// TwinCAT 3 PLC project Lectures
// ProgramVersion: 3.1.4024.0
// libraries:
//   Tc2_Standard, * (Beckhoff Automation GmbH)
//   Tc2_System, * (Beckhoff Automation GmbH)
//   Tc3_Module, * (Beckhoff Automation GmbH)
// project tree:
//   DUTs/ Item.TcDUT (not stored), Location.TcDUT
//   GVLs/ Automatic.TcGVL, IO.TcGVL
//   / PlcTask.TcTTO
//   POUs/ AutomaticControl.TcPOU, CountCurrentPosition.TcPOU, CountCurrentPosition1.TcPOU, Initialize.TcPOU, ManualControl.TcPOU, MAIN.TcPOU, Motor.TcPOU, MotorSelection.TcPOU, Recipe1.TcPOU, Recipe11.TcPOU, Recipe13.TcPOU, Recipe2.TcPOU, RestorePreviousAutomaticState.TcPOU, Safety1.TcPOU (not stored)
//   POUs/Lectures%27 programs/ p00_true_false.TcPOU (not stored), p01_sequential.TcPOU (not stored), p02_clock.TcPOU (not stored), p03_SR1.TcPOU (not stored), p04_latch.TcPOU (not stored), p05_posEdge.TcPOU (not stored), p06_frontDetection.TcPOU (not stored), p07_memoryCell.TcPOU (not stored), p08_counter.TcPOU (not stored), p09_timers.TcPOU (not stored), p10_directionalInterlock.TcPOU (not stored), p11_logicalFunction.TcPOU (not stored), p12_controlLight.TcPOU (not stored)
// real-time tasks:
//   TASK PlcTask1: cycle T#10ms, priority 21, ADS port 351
//   TASK PlcTask: cycle T#10ms, priority 20, ADS port 350
// I/O:
//   DEVICE Device 1 (EtherCAT), AmsNetId 172.31.192.1.2.1
//     Term 1 (EK1200) [EK1200-7000 EtherCAT Power supply (1,5A E-Bus)]
//       Term 2 (EL1859) [EL1859 8Ch. Dig. Input 24V, 3ms, 8Ch. Dig. Output 24V, 0.5A]
//       Term 3 (EL1859) [EL1859 8Ch. Dig. Input 24V, 3ms, 8Ch. Dig. Output 24V, 0.5A]
//       Term 4 (EL9011) [EL9011 End Terminal]
//   DEVICE Device 2 (NOV-DP-RAM) (disabled)
//   DEVICE Device 3 (CX7000), AmsNetId 172.31.192.1.4.1
//     Term 1 (CX7028) [CX7028-0000-0121]
//       modules: Module 1 (DIO_2x), Module 2 (Empty Module), Module 3 (DIO_2x), Module 4 (Empty Module), Module 5 (DI_2x), Module 6 (Empty Module), Module 7 (DI_2x), Module 8 (Empty Module)
// variable links:
//   Lectures/Lectures Instance <-> Device 1 (EtherCAT)/Term 1 (EK1200)/Term 2 (EL1859)
//     PlcTask Inputs/IO.EndExtensionSensor <-> Channel 3/Input
//     PlcTask Inputs/IO.EndGripSensor <-> Channel 7/Input
//     PlcTask Inputs/IO.EndLiftingSensor <-> Channel 5/Input
//     PlcTask Inputs/IO.EndRotationSensor <-> Channel 1/Input
//     PlcTask Inputs/IO.StepExtensionSwitch <-> Channel 4/Input
//     PlcTask Inputs/IO.StepGripSwitch <-> Channel 8/Input
//     PlcTask Inputs/IO.StepLiftingSwitch <-> Channel 6/Input
//     PlcTask Inputs/IO.StepRotatonSwitch <-> Channel 2/Input
//     PlcTask Outputs/IO.MotorExtension <-> Channel 12/Output
//     PlcTask Outputs/IO.MotorExtensionDirection <-> Channel 11/Output
//     PlcTask Outputs/IO.MotorGrip <-> Channel 16/Output
//     PlcTask Outputs/IO.MotorGripDirection <-> Channel 15/Output
//     PlcTask Outputs/IO.MotorLifting <-> Channel 14/Output
//     PlcTask Outputs/IO.MotorLiftingDirection <-> Channel 13/Output
//     PlcTask Outputs/IO.MotorRotation <-> Channel 10/Output
//     PlcTask Outputs/IO.MotorRotationDirection <-> Channel 9/Output
//   Lectures/Lectures Instance <-> Device 3 (CX7000)/Term 1 (CX7028)
//     PlcTask Inputs/IO.ButtonGreen <-> Module 3 (DIO_2x)/DIO_2x Input Channel 2/Input
//     PlcTask Inputs/IO.ButtonLowerLeft <-> Module 5 (DI_2x)/DI_2x Input Channel 1/Input
//     PlcTask Inputs/IO.ButtonLowerRight <-> Module 5 (DI_2x)/DI_2x Input Channel 2/Input
//     PlcTask Inputs/IO.ButtonRed <-> Module 1 (DIO_2x)/DIO_2x Input Channel 1/Input
//     PlcTask Inputs/IO.ButtonUpperLeft <-> Module 1 (DIO_2x)/DIO_2x Input Channel 2/Input
//     PlcTask Inputs/IO.ButtonUpperRight <-> Module 3 (DIO_2x)/DIO_2x Input Channel 1/Input
//     PlcTask Inputs/IO.Switch <-> Module 7 (DI_2x)/DI_2x Input Channel 1/Input
//     PlcTask Outputs/IO.LEDBlueLower <-> Module 3 (DIO_2x)/DIO_2x Output Channel 2/Output
//     PlcTask Outputs/IO.LEDBlueUpper <-> Module 1 (DIO_2x)/DIO_2x Output Channel 2/Output
//     PlcTask Outputs/IO.LEDGreen <-> Module 3 (DIO_2x)/DIO_2x Output Channel 1/Output
//     PlcTask Outputs/IO.LEDRed <-> Module 1 (DIO_2x)/DIO_2x Output Channel 1/Output

CONFIGURATION Lectures
    RESOURCE PLC ON TwinCAT3
        TASK PlcTask(INTERVAL := T#10ms, PRIORITY := 21);
        PROGRAM MAIN WITH PlcTask : MAIN;
    END_RESOURCE
END_CONFIGURATION

// ---- DUTs/Location.TcDUT
TYPE Location:
STRUCT
	rotation: REAL;	// need to get full circle number...
	lifting: REAL;	// need to get the full lift number...
	extension: REAL; // need to get the full extension number...
	grip: REAL;	// need to get the full grip number...
END_STRUCT
END_TYPE

// ---- GVLs/Automatic.TcGVL
{attribute 'qualified_only'}
VAR_GLOBAL
	MotorR: Motor;
	RCurrentlyMoving: BOOL;
	RotationPositionAuto: INT;
	RotationPositionCurrent: INT;
	SafetyRON: BOOL;
	
	MotorL: Motor;
	LCurrentlyMoving: BOOL;
	LiftingPositionAuto: INT;
	LiftingPositionCurrent: INT;
	SafetyLON: BOOL;
	
	MotorE: Motor;
	ECurrentlyMoving: BOOL;
	ExtensionPositionAuto: INT;
	ExtensionPositionCurrent: INT;
	SafetyEON: BOOL;
	
	MotorG: Motor;
	GCurrentlyMoving: BOOL;
	GripPositionAuto: INT;
	GripPositionCurrent: INT;
	SafetyGON: BOOL;
	
	AllRestored: BOOL;
END_VAR

// ---- GVLs/IO.TcGVL
{attribute 'qualified_only'}
VAR_GLOBAL
	ButtonRed AT %I*: BOOL;
	ButtonUpperRight AT %I*: BOOL;
	ButtonLowerLeft AT %I*: BOOL;
	Switch AT %I*: BOOL;
	LEDRed AT %Q*: BOOL;
	LEDGreen AT %Q*: BOOL;
	ButtonUpperLeft AT %I*: BOOL;
	ButtonGreen AT %I*: BOOL;
	ButtonLowerRight AT %I*: BOOL;
	LEDBlueUpper AT %Q*: BOOL;
	LEDBlueLower AT %Q*: BOOL;
	
	EndRotationSensor AT %I*: BOOL;
	StepRotatonSwitch AT %I*: BOOL;
	EndExtensionSensor AT %I*: BOOL;
	StepExtensionSwitch AT %I*: BOOL;
	EndLiftingSensor AT %I*: BOOL;
	StepLiftingSwitch AT %I*: BOOL;
	EndGripSensor AT %I*: BOOL;
	StepGripSwitch AT %I*: BOOL;
	MotorRotationDirection AT %Q*: BOOL;
	MotorRotation AT %Q*: BOOL;
	MotorExtensionDirection AT %Q*: BOOL;
	MotorExtension AT %Q*: BOOL;
	MotorLiftingDirection AT %Q*: BOOL;
	MotorLifting AT %Q*: BOOL;
	MotorGripDirection AT %Q*: BOOL;
	MotorGrip AT %Q*: BOOL;
	Initialized: BOOL;
	MotorDirection: INT;
	PreviousManualMode: BOOL;
END_VAR

// ---- POUs/MAIN.TcPOU
PROGRAM MAIN
VAR
	ManualControl_0: ManualControl;
	AutomaticControl_0: AutomaticControl;
END_VAR

// Initially it goes to position (0,0,0,0) and initializes motors by Initialize PRG.
// There is Safety PRG that keeps checking if motors are out of bounds.
// Motors are instantiated as global vars to retain their properties.
// CountCurrentPosition PRG is the only place where we count position using the sensors.
// RestorePreviousAutomaticState is a FB that gets execture cyclic until all the directions are set to previous positions.
// AutomaticControl FB remembers which recipe is being executed and recipe remembers its state.

// TODO:
// delay...
// ce ne dela zakomentiraj Safety
VAR // added by the converter: edge detectors and wires of the graphical bodies
    _ft1 : F_TRIG;
    _rt1 : R_TRIG;
    _w1 : BOOL;
END_VAR

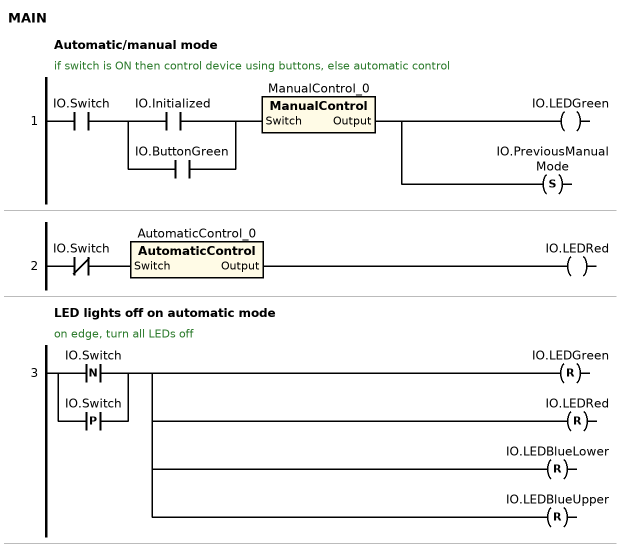
// NETWORK 1: Automatic/manual mode
// if switch is ON then control device using buttons, else automatic control
ManualControl_0(Switch := IO.Switch AND IO.Initialized OR IO.Switch AND IO.ButtonGreen); // ManualControl
IO.LEDGreen := ManualControl_0.Output;
IO.PreviousManualMode S= ManualControl_0.Output;

// NETWORK 2
AutomaticControl_0(Switch := NOT IO.Switch); // AutomaticControl
IO.LEDRed := AutomaticControl_0.Output;

// NETWORK 3: LED lights off on automatic mode
// on edge, turn all LEDs off
_ft1(CLK := IO.Switch);
_rt1(CLK := IO.Switch);
_w1 := _ft1.Q OR _rt1.Q;
IO.LEDGreen R= _w1;
IO.LEDRed R= _w1;
IO.LEDBlueLower R= _w1;
IO.LEDBlueUpper R= _w1;

END_PROGRAM

// ---- POUs/ManualControl.TcPOU
FUNCTION_BLOCK PUBLIC ManualControl
VAR_INPUT
	Switch: BOOL;
END_VAR
VAR
	ManualControl: BOOL;
	TimeForInterlockDelay: TIME := T#0.05S;
	ManualMode: BOOL;
	MotorSelection_1: MotorSelection;
	SelectedMotor: INT;
	temp: TIME;
	LowerLeftInterlock: TOF;
	LowerLeft: BOOL;
	LowerRightInterlock: TOF;
	LowerRight: BOOL;
END_VAR
VAR_OUTPUT
	Output: BOOL;
END_VAR
VAR // added by the converter: edge detectors and wires of the graphical bodies
    _w1, _w2, _w3, _w4, _w5, _w6, _w7, _w8, _w9, _w10, _w11, _w12 : BOOL;
    _rt1, _rt2, _rt3, _rt4 : R_TRIG;
    _ft1, _ft2, _ft3, _ft4 : F_TRIG;
END_VAR

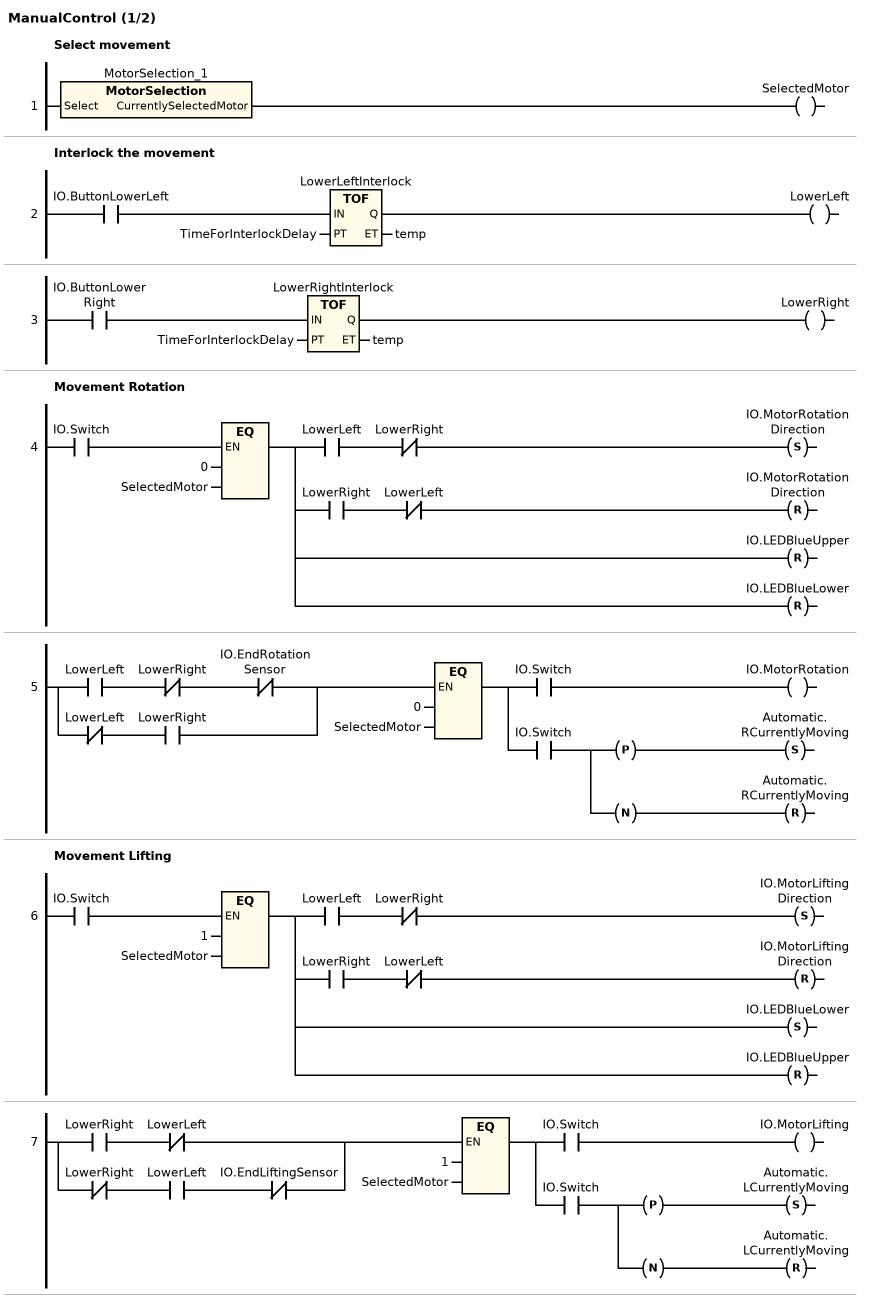
// NETWORK 1: Select movement
MotorSelection_1(Select := TRUE); // MotorSelection
SelectedMotor := MotorSelection_1.CurrentlySelectedMotor;

// NETWORK 2: Interlock the movement
LowerLeftInterlock(IN := IO.ButtonLowerLeft, PT := TimeForInterlockDelay, ET => temp); // TOF
LowerLeft := LowerLeftInterlock.Q;

// NETWORK 3
LowerRightInterlock(IN := IO.ButtonLowerRight, PT := TimeForInterlockDelay, ET => temp); // TOF
LowerRight := LowerRightInterlock.Q;

// NETWORK 4: Movement Rotation
_w1 := IO.Switch AND 0 = SelectedMotor;
IO.MotorRotationDirection S= _w1 AND LowerLeft AND NOT LowerRight;
IO.MotorRotationDirection R= _w1 AND LowerRight AND NOT LowerLeft;
IO.LEDBlueUpper R= _w1;
IO.LEDBlueLower R= _w1;

// NETWORK 5
_w2 := (LowerLeft AND NOT LowerRight AND NOT IO.EndRotationSensor OR NOT LowerLeft AND LowerRight) AND 0 = SelectedMotor;
IO.MotorRotation := _w2 AND IO.Switch;
_w3 := _w2 AND IO.Switch;
_rt1(CLK := _w3);
Automatic.RCurrentlyMoving S= _rt1.Q;
_ft1(CLK := _w3);
Automatic.RCurrentlyMoving R= _ft1.Q;

// NETWORK 6: Movement Lifting
_w4 := IO.Switch AND 1 = SelectedMotor;
IO.MotorLiftingDirection S= _w4 AND LowerLeft AND NOT LowerRight;
IO.MotorLiftingDirection R= _w4 AND LowerRight AND NOT LowerLeft;
IO.LEDBlueLower S= _w4;
IO.LEDBlueUpper R= _w4;

// NETWORK 7
_w5 := (LowerRight AND NOT LowerLeft OR NOT LowerRight AND LowerLeft AND NOT IO.EndLiftingSensor) AND 1 = SelectedMotor;
IO.MotorLifting := _w5 AND IO.Switch;
_w6 := _w5 AND IO.Switch;
_rt2(CLK := _w6);
Automatic.LCurrentlyMoving S= _rt2.Q;
_ft2(CLK := _w6);
Automatic.LCurrentlyMoving R= _ft2.Q;

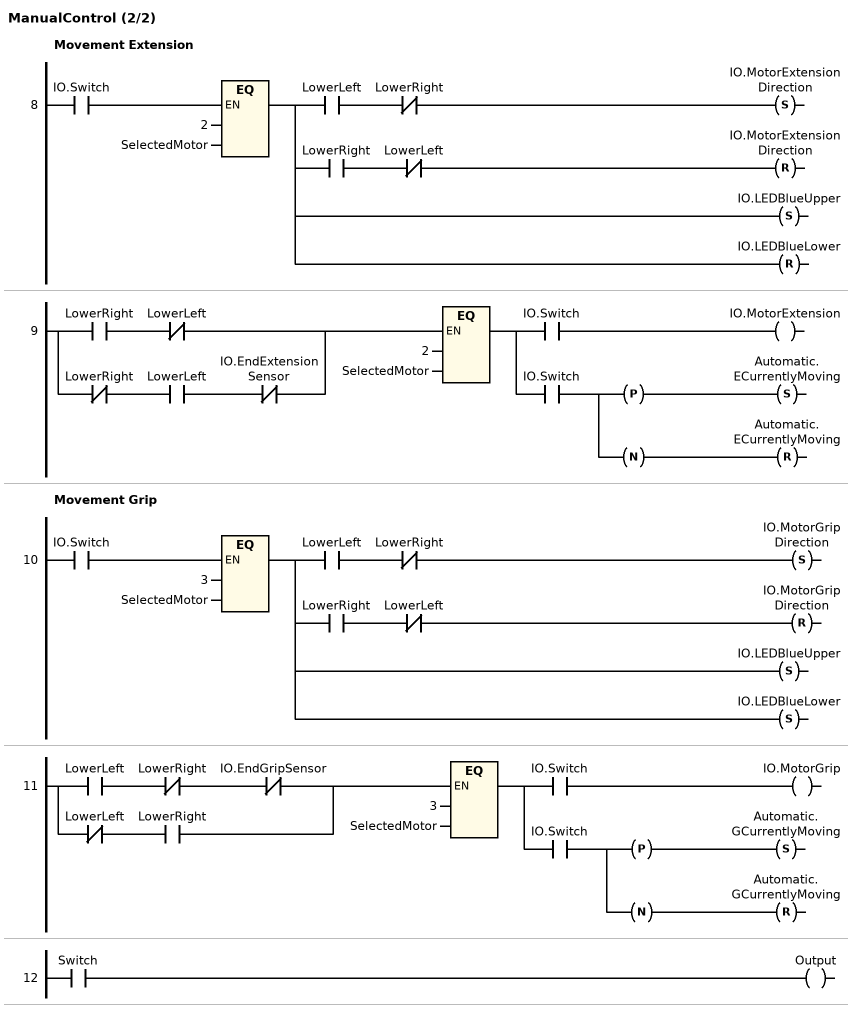
// NETWORK 8: Movement Extension
_w7 := IO.Switch AND 2 = SelectedMotor;
IO.MotorExtensionDirection S= _w7 AND LowerLeft AND NOT LowerRight;
IO.MotorExtensionDirection R= _w7 AND LowerRight AND NOT LowerLeft;
IO.LEDBlueUpper S= _w7;
IO.LEDBlueLower R= _w7;

// NETWORK 9
_w8 := (LowerRight AND NOT LowerLeft OR NOT LowerRight AND LowerLeft AND NOT IO.EndExtensionSensor) AND 2 = SelectedMotor;
IO.MotorExtension := _w8 AND IO.Switch;
_w9 := _w8 AND IO.Switch;
_rt3(CLK := _w9);
Automatic.ECurrentlyMoving S= _rt3.Q;
_ft3(CLK := _w9);
Automatic.ECurrentlyMoving R= _ft3.Q;

// NETWORK 10: Movement Grip
_w10 := IO.Switch AND 3 = SelectedMotor;
IO.MotorGripDirection S= _w10 AND LowerLeft AND NOT LowerRight;
IO.MotorGripDirection R= _w10 AND LowerRight AND NOT LowerLeft;
IO.LEDBlueUpper S= _w10;
IO.LEDBlueLower S= _w10;

// NETWORK 11
_w11 := (LowerLeft AND NOT LowerRight AND NOT IO.EndGripSensor OR NOT LowerLeft AND LowerRight) AND 3 = SelectedMotor;
IO.MotorGrip := _w11 AND IO.Switch;
_w12 := _w11 AND IO.Switch;
_rt4(CLK := _w12);
Automatic.GCurrentlyMoving S= _rt4.Q;
_ft4(CLK := _w12);
Automatic.GCurrentlyMoving R= _ft4.Q;

// NETWORK 12
Output := Switch;

END_FUNCTION_BLOCK

// ---- POUs/MotorSelection.TcPOU
FUNCTION_BLOCK PUBLIC MotorSelection
VAR_INPUT
	Select: BOOL;
END_VAR
VAR
	TimeForDelay: TIME := T#0.15S;
	MovementSelection: CTUD;
	SelectionCounter: CTUD := (LOAD := TRUE, PV := 3);
	ReachedMaxSelection: BOOL;
	ReachedMinSelection: BOOL;
	UpperLeftDelay: TOF;
	UpperRightDelay: TOF;
	tmnp: TIME;
	CU: BOOL;
	CD: BOOL;
	CUU: BOOL;
	CDD: BOOL;
	PositiveEdge1: R_TRIG;
	PositiveEdge2: R_TRIG;
	temporary: BOOL;
	CUU0: BOOL;
	CDD0: BOOL;
	temporary1: BOOL;
	BURpositiveEdge: BOOL;
	BULpositiveEdge: BOOL;
	temp2: BOOL;
	temp3: BOOL;
END_VAR
VAR_OUTPUT
	CurrentlySelectedMotor: INT;
END_VAR
VAR // added by the converter: edge detectors and wires of the graphical bodies
    _rt1, _rt2, _rt3, _rt4 : R_TRIG;
END_VAR

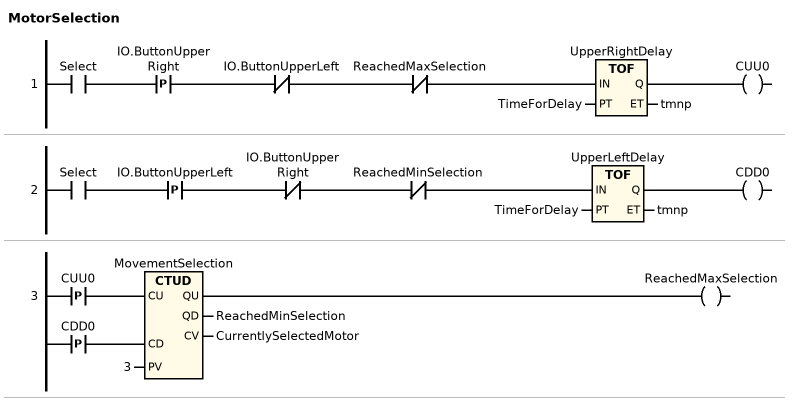
// NETWORK 1
_rt1(CLK := IO.ButtonUpperRight);
UpperRightDelay(
    IN := Select AND _rt1.Q AND NOT IO.ButtonUpperLeft AND NOT ReachedMaxSelection,
    PT := TimeForDelay,
    ET => tmnp); // TOF
CUU0 := UpperRightDelay.Q;

// NETWORK 2
_rt2(CLK := IO.ButtonUpperLeft);
UpperLeftDelay(
    IN := Select AND _rt2.Q AND NOT IO.ButtonUpperRight AND NOT ReachedMinSelection,
    PT := TimeForDelay,
    ET => tmnp); // TOF
CDD0 := UpperLeftDelay.Q;

// NETWORK 3
_rt3(CLK := CUU0);
_rt4(CLK := CDD0);
MovementSelection(
    CU := _rt3.Q,
    CD := _rt4.Q,
    PV := 3,
    QD => ReachedMinSelection,
    CV => CurrentlySelectedMotor); // CTUD
ReachedMaxSelection := MovementSelection.QU;

END_FUNCTION_BLOCK

// ---- POUs/AutomaticControl.TcPOU
FUNCTION_BLOCK PUBLIC AutomaticControl
VAR_INPUT
    Switch: BOOL;
END_VAR
VAR
    State: INT := 0;
    ExecutingRecipe1: BOOL := FALSE;
    ExecutingRecipe2: BOOL := FALSE;
    myRecipe2: Recipe2;
    Tmp: BOOL;
    RestorePreviousAutomaticState: RestorePreviousAutomaticState;
	CountCurrentPosition1: CountCurrentPosition1;
	Safety: Safety1;
END_VAR
VAR_OUTPUT
    Output: BOOL := TRUE;
END_VAR

// TwinCAT ensures that all POUs, including your AutomaticControl program 
// and Recipe1() Function Block, are executed once per cycle.

IF NOT IO.Initialized THEN
	Initialize();
ELSIF NOT IO.Switch AND IO.PreviousManualMode THEN
	Automatic.AllRestored := FALSE;
	CountCurrentPosition1();
    RestorePreviousAutomaticState();
	Safety();
ELSE
	CountCurrentPosition1();
	Safety();
	
    IF (IO.ButtonUpperLeft OR ExecutingRecipe1) AND Automatic.AllRestored THEN
		//Automatic.AllRestored := FALSE;
        ExecutingRecipe1 := TRUE;
		Recipe1();
        ExecutingRecipe1 := NOT Recipe1.SuccesfullyEnded; // Update ExecutingRecipe1 based on output
    ELSIF NOT ExecutingRecipe1 AND (IO.ButtonUpperRight OR ExecutingRecipe2) THEN
        ExecutingRecipe2 := TRUE;
        myRecipe2.ExecutingRecipe2 := ExecutingRecipe2; // Pass input to the function block
        //myRecipe2(); // Call the function block
        ExecutingRecipe2 := NOT myRecipe2.SuccesfullyEnded; // Update ExecutingRecipe2 based on output
    END_IF
END_IF


// for debugging purposes:
IF IO.ButtonRed THEN
	IO.Initialized := FALSE;
END_IF

RETURN;

END_FUNCTION_BLOCK

// ---- POUs/Recipe2.TcPOU
FUNCTION_BLOCK PUBLIC Recipe2
VAR_INPUT
	ExecutingRecipe2: BOOL;
END_VAR
VAR_OUTPUT
	SuccesfullyEnded: BOOL := FALSE;
END_VAR
VAR
	State: INT := 0;
	InitialRotationPosition: INT := 140;
	InitialLiftingPosition: INT := 200;
	MaxGripPosition: INT := 160;
END_VAR

// Recipe is sequence of moves to execute the task.

IF ExecutingRecipe2 THEN	// we start executing recipe2 (again)
	SuccesfullyEnded := FALSE;
END_IF

IF NOT IO.Switch AND NOT SuccesfullyEnded THEN
	// WOOD:
	IF State = 0 THEN
		IF Automatic.RotationPositionAuto < InitialRotationPosition THEN
			IO.MotorRotationDirection := 0;
			IF NOT Automatic.SafetyRON THEN
				Automatic.MotorR.CurrentlyMoving := TRUE;
				IO.MotorRotation := 1;
			END_IF
		ELSE
			State := 1;
			IO.MotorRotation := 0;
			Automatic.MotorR.CurrentlyMoving := FALSE;
		END_IF
	ELSIF State = 1 THEN
		IF Automatic.LiftingPositionAuto < InitialLiftingPosition THEN
			IO.MotorLiftingDirection := 1;
			IF NOT Automatic.SafetyLON THEN
				Automatic.MotorL.CurrentlyMoving := TRUE;
				IO.MotorLifting := 1;
			END_IF
		ELSE
			State := 2;
			IO.MotorLifting := 0;
			Automatic.MotorL.CurrentlyMoving := FALSE;
		END_IF
	ELSIF State = 2 THEN
		IF Automatic.GripPositionAuto < MaxGripPosition THEN
			IO.MotorGripDirection := 0;
			IF NOT Automatic.SafetyGON THEN
				Automatic.MotorG.CurrentlyMoving := TRUE;
				IO.MotorGrip := 1;
			END_IF
		ELSE
			State := 3;
			IO.MotorGrip := 0;
			Automatic.MotorG.CurrentlyMoving := FALSE;
		END_IF
	ELSIF State = 3 THEN
		IF NOT IO.EndLiftingSensor THEN
			IO.MotorLiftingDirection := 0;
			IF NOT Automatic.SafetyLON THEN
				Automatic.MotorG.CurrentlyMoving := TRUE;
				IO.MotorLifting := 1;
			END_IF
		ELSE
			State := 4;
			IO.MotorLifting := 0;
			Automatic.MotorG.CurrentlyMoving := FALSE;
		END_IF
	ELSIF State = 4 THEN
		IF NOT IO.EndRotationSensor THEN
			IO.MotorRotationDirection := 1;
			IF NOT Automatic.SafetyRON THEN
				Automatic.MotorR.CurrentlyMoving := TRUE;
				IO.MotorRotation := 1;
			END_IF
		ELSE
			State := 5;
			IO.MotorRotation := 0;
			Automatic.MotorR.CurrentlyMoving := FALSE;
		END_IF
	ELSIF State = 5 THEN
		IF NOT IO.EndGripSensor THEN		// it places the cylinder onto the platform
			IO.MotorGripDirection := 1;
			IF NOT Automatic.SafetyGON THEN
				Automatic.MotorG.CurrentlyMoving := TRUE;
				IO.MotorGrip := 1;
			END_IF
		ELSE
			State := 6;
			IO.MotorGrip := 0;
			Automatic.MotorG.CurrentlyMoving := FALSE;
		END_IF
	ELSIF State = 6 THEN
		SuccesfullyEnded := TRUE;
		State := 0;
		RETURN;
	END_IF
END_IF

END_FUNCTION_BLOCK

// ---- POUs/RestorePreviousAutomaticState.TcPOU
FUNCTION_BLOCK PUBLIC RestorePreviousAutomaticState
VAR_INPUT
END_VAR
VAR_OUTPUT
END_VAR
VAR
	RotationRestored: BOOL := FALSE;
	LiftingRestored: BOOL := FALSE;
	ExtensionRestored: BOOL := FALSE;
	GripRestored: BOOL := FALSE;
END_VAR

// reset rotation:
IO.LEDRed := 1;
IF Automatic.RotationPositionAuto - Automatic.RotationPositionCurrent > 5 AND NOT RotationRestored AND NOT Automatic.SafetyRON THEN
	IO.MotorRotationDirection := 0;
	Automatic.RCurrentlyMoving := TRUE;
	IO.MotorRotation := 1;
ELSIF Automatic.RotationPositionCurrent - Automatic.RotationPositionAuto > 5 AND NOT RotationRestored AND NOT Automatic.SafetyRON THEN
	IO.MotorRotationDirection := 1;
	Automatic.RCurrentlyMoving := TRUE;
	IO.MotorRotation := 1;
ELSE
	Automatic.RCurrentlyMoving := FALSE;
	IO.MotorRotation := 0;
	RotationRestored := TRUE;
END_IF

// reset lifting:
IF Automatic.LiftingPositionAuto - Automatic.LiftingPositionCurrent > 5 AND NOT LiftingRestored AND NOT Automatic.SafetyLON THEN
	IO.MotorLiftingDirection := 0;
	Automatic.LCurrentlyMoving := TRUE;
	IO.MotorLifting := 1;
ELSIF Automatic.LiftingPositionCurrent - Automatic.LiftingPositionAuto > 5 AND NOT LiftingRestored AND NOT Automatic.SafetyLON THEN
	IO.MotorLiftingDirection := 0;
	Automatic.LCurrentlyMoving := TRUE;
	IO.MotorLifting := 1;
ELSE
	Automatic.LCurrentlyMoving := FALSE;
	IO.MotorLifting := 0;
	LiftingRestored := TRUE;
END_IF

// reset extension:
IF Automatic.ExtensionPositionAuto - Automatic.ExtensionPositionCurrent > 5 AND NOT ExtensionRestored AND NOT Automatic.SafetyEON THEN
	IO.MotorExtensionDirection := 0;
	Automatic.ECurrentlyMoving := TRUE;
	IO.MotorExtension := 1;
ELSIF Automatic.ExtensionPositionCurrent - Automatic.ExtensionPositionAuto > 5 AND NOT ExtensionRestored AND NOT Automatic.SafetyEON THEN
	IO.MotorExtensionDirection := 0;
	Automatic.ECurrentlyMoving := TRUE;
	IO.MotorExtension := 1;
ELSE
	Automatic.ECurrentlyMoving := FALSE;
	IO.MotorExtension := 0;
	ExtensionRestored := TRUE;
END_IF

// reset grip:
IF Automatic.GripPositionAuto - Automatic.GripPositionCurrent > 5 AND NOT GripRestored AND NOT Automatic.SafetyGON THEN
	IO.MotorGripDirection := 0;
	Automatic.GCurrentlyMoving := TRUE;
	IO.MotorGrip := 1;
ELSIF Automatic.GripPositionCurrent - Automatic.GripPositionAuto > 5 AND NOT GripRestored AND NOT Automatic.SafetyGON THEN
	IO.MotorGripDirection := 0;
	Automatic.GCurrentlyMoving := TRUE;
	IO.MotorGrip := 1;
ELSE
	Automatic.GCurrentlyMoving := FALSE;
	IO.MotorGrip := 0;
	GripRestored := TRUE;
END_IF

// if all restored then go on to exeecute recipes in AutomaticControl:
IF RotationRestored AND LiftingRestored AND ExtensionRestored AND GripRestored THEN
	IO.LEDRed := 0;
	IO.PreviousManualMode := FALSE;
	Automatic.AllRestored := TRUE;
	RotationRestored := FALSE;
	ExtensionRestored := FALSE;
	LiftingRestored := FALSE;
	GripRestored := FALSE;
	Automatic.RCurrentlyMoving := FALSE;
	Automatic.ECurrentlyMoving := FALSE;
	Automatic.LCurrentlyMoving := FALSE;
	Automatic.GCurrentlyMoving := FALSE;
END_IF

END_FUNCTION_BLOCK

// ---- POUs/CountCurrentPosition1.TcPOU
FUNCTION_BLOCK CountCurrentPosition1
VAR_INPUT
END_VAR
VAR_OUTPUT
END_VAR
VAR
END_VAR

// COUNT ROTATION:
IF IO.Initialized AND IO.StepRotatonSwitch = 1 THEN
	IF IO.MotorRotationDirection = 0 THEN
		IF (NOT IO.Switch) AND Automatic.RCurrentlyMoving THEN
			IF IO.PreviousManualMode THEN
				Automatic.RotationPositionCurrent := Automatic.RotationPositionCurrent + 1;
			ELSE
				Automatic.RotationPositionCurrent := Automatic.RotationPositionCurrent + 1;
				Automatic.RotationPositionAuto := Automatic.RotationPositionAuto + 1;
			END_IF
		ELSIF Automatic.RCurrentlyMoving THEN
			Automatic.RotationPositionCurrent := Automatic.RotationPositionCurrent + 1;
		END_IF
	ELSE
		IF (NOT IO.Switch) AND Automatic.RCurrentlyMoving THEN
			IF IO.PreviousManualMode THEN
				Automatic.RotationPositionCurrent := Automatic.RotationPositionCurrent - 1;
			ELSE
				Automatic.RotationPositionCurrent := Automatic.RotationPositionCurrent - 1;
				Automatic.RotationPositionAuto := Automatic.RotationPositionAuto - 1;
			END_IF
		ELSIF Automatic.RCurrentlyMoving THEN
			Automatic.RotationPositionCurrent := Automatic.RotationPositionCurrent - 1;
		END_IF
	END_IF
END_IF

// COUNT Extension:
IF IO.Initialized AND IO.StepExtensionSwitch = 1 THEN
	IO.LEDGreen := 0;
	IF IO.MotorExtensionDirection = 0 THEN
		IF (NOT IO.Switch) AND Automatic.ECurrentlyMoving THEN
			IF IO.PreviousManualMode THEN
				Automatic.ExtensionPositionCurrent := Automatic.ExtensionPositionCurrent + 1;
			ELSE
				Automatic.ExtensionPositionAuto := Automatic.ExtensionPositionAuto + 1;
				Automatic.ExtensionPositionCurrent := Automatic.ExtensionPositionCurrent + 1;
			END_IF
		ELSIF Automatic.ECurrentlyMoving THEN
			Automatic.ExtensionPositionCurrent := Automatic.ExtensionPositionCurrent + 1;
		END_IF
	ELSE
		IF (NOT IO.Switch) AND Automatic.ECurrentlyMoving THEN
			IF IO.PreviousManualMode THEN
				Automatic.ExtensionPositionCurrent := Automatic.ExtensionPositionCurrent - 1;
			ELSE
				Automatic.ExtensionPositionAuto := Automatic.ExtensionPositionAuto - 1;
				Automatic.ExtensionPositionCurrent := Automatic.ExtensionPositionCurrent - 1;
			END_IF
		ELSIF Automatic.ECurrentlyMoving THEN
			Automatic.ExtensionPositionCurrent := Automatic.ExtensionPositionCurrent - 1;
		END_IF
	END_IF
END_IF

// COUNT Lifting:
IF IO.Initialized AND IO.StepLiftingSwitch = 1 THEN
	IF IO.MotorLiftingDirection = 0 THEN
		IF (NOT IO.Switch) AND Automatic.LCurrentlyMoving THEN
			IF IO.PreviousManualMode THEN
				Automatic.LiftingPositionCurrent := Automatic.LiftingPositionCurrent + 1;
			ELSE
				Automatic.LiftingPositionCurrent := Automatic.LiftingPositionCurrent + 1;
				Automatic.LiftingPositionAuto := Automatic.LiftingPositionAuto + 1;
			END_IF
		ELSIF Automatic.LCurrentlyMoving THEN
			Automatic.LiftingPositionCurrent := Automatic.LiftingPositionCurrent + 1;
		END_IF
	ELSE
		IF (NOT IO.Switch) AND Automatic.LCurrentlyMoving THEN
			IF IO.PreviousManualMode THEN
				Automatic.LiftingPositionCurrent := Automatic.LiftingPositionCurrent - 1;
			ELSE
				Automatic.LiftingPositionAuto := Automatic.LiftingPositionAuto - 1;
				Automatic.LiftingPositionCurrent := Automatic.LiftingPositionCurrent - 1;
			END_IF
		ELSIF Automatic.LCurrentlyMoving THEN
			Automatic.LiftingPositionCurrent := Automatic.LiftingPositionCurrent - 1;
		END_IF
	END_IF
END_IF

// COUNT Grip:
IF IO.Initialized AND IO.StepGripSwitch = 1 THEN
	IF IO.MotorGripDirection = 0 THEN
		IF (NOT IO.Switch) AND Automatic.GCurrentlyMoving THEN	// automatic mode
			IO.LEDGreen := 0;
			
			IF IO.PreviousManualMode THEN
				Automatic.GripPositionCurrent := Automatic.GripPositionCurrent + 1;
			ELSE
				Automatic.GripPositionAuto := Automatic.GripPositionAuto + 1;
				Automatic.GripPositionCurrent := Automatic.GripPositionCurrent + 1;
			END_IF
		ELSIF Automatic.GCurrentlyMoving THEN		// manual mode
			Automatic.GripPositionCurrent := Automatic.GripPositionCurrent + 1;
		END_IF
	ELSE
		IF (NOT IO.Switch) AND Automatic.GCurrentlyMoving THEN
			IO.LEDGreen := 1;
			IF IO.PreviousManualMode THEN
				Automatic.GripPositionCurrent := Automatic.GripPositionCurrent - 1;
			ELSE
				Automatic.GripPositionAuto := Automatic.GripPositionAuto - 1;
				Automatic.GripPositionCurrent := Automatic.GripPositionCurrent - 1;
			END_IF
		ELSIF Automatic.GCurrentlyMoving THEN
			Automatic.GripPositionCurrent := Automatic.GripPositionCurrent - 1;
		END_IF
	END_IF
END_IF

END_FUNCTION_BLOCK

// ---- POUs/Initialize.TcPOU
PROGRAM Initialize
VAR
END_VAR

// go to the initial position (0,0,0,0)
IF NOT IO.Initialized THEN
	IF IO.EndRotationSensor THEN
		IO.MotorRotation := 0;
		IO.MotorRotationDirection := 0;
		Automatic.MotorR.CurrentlyMoving := FALSE;
	ELSE 
		IO.MotorRotationDirection := 1;
		Automatic.MotorR.CurrentlyMoving := TRUE;
		IO.MotorRotation := 1;
	END_IF
	
	IF IO.EndLiftingSensor THEN
		IO.MotorLifting := 0;
		IO.MotorLiftingDirection := 0;
		Automatic.MotorL.CurrentlyMoving := FALSE;
	ELSE 
		IO.MotorLiftingDirection := 1;
		Automatic.MotorL.CurrentlyMoving := TRUE;
		IO.MotorLifting := 1;
	END_IF
	
	IF IO.EndExtensionSensor THEN
		IO.MotorExtension := 0;
		IO.MotorExtensionDirection := 0;
		Automatic.MotorE.CurrentlyMoving := FALSE;
	ELSE 
		IO.MotorExtensionDirection := 1;
		Automatic.MotorE.CurrentlyMoving := TRUE;
		IO.MotorExtension := 1;
	END_IF
	
	IF IO.EndGripSensor THEN
		IO.MotorGrip := 0;
		IO.MotorGripDirection := 0;
		Automatic.MotorG.CurrentlyMoving := FALSE;
	ELSE 
		IO.MotorGripDirection := 1;
		Automatic.MotorG.CurrentlyMoving := TRUE;
		IO.MotorGrip := 1;
	END_IF
		
	IF IO.EndRotationSensor AND IO.EndLiftingSensor AND IO.EndExtensionSensor AND IO.EndGripSensor THEN
		Automatic.MotorR.CurrentlyMoving := FALSE;
		Automatic.MotorE.CurrentlyMoving := FALSE;
		Automatic.MotorL.CurrentlyMoving := FALSE;
		Automatic.MotorG.CurrentlyMoving := FALSE;
		IO.Initialized := TRUE;
	END_IF
END_IF

END_PROGRAM

// ---- POUs/Recipe1.TcPOU
FUNCTION_BLOCK PUBLIC Recipe1
VAR_INPUT
	ExecutingRecipe1: BOOL;
END_VAR
VAR_OUTPUT
	SuccesfullyEnded: BOOL := FALSE;
END_VAR
VAR
	State: INT := 0;
	WoodInitialLiftingPosition: INT := 50;
	InitialExtensionPosition: INT := 388;
	MaxGripPosition: INT := 160;
	RotationDropOffPosition: INT := 300;
	PlasticsInitialLiftingPosition: INT := 250;
	PlasticsDropOffExtensionPosition: INT := 300;
	MetalInitialLiftingPosition: INT := 400;
	MetalDropOffExtensionPosition: INT := 500;
END_VAR

// Recipe is sequence of moves to execute the task.

IF ExecutingRecipe1 THEN	// we start executing recipe1 (again)
	SuccesfullyEnded := FALSE;
END_IF

IF NOT IO.Switch AND NOT SuccesfullyEnded THEN
	// WOOD:
	IF State = 0 THEN
		IF Automatic.LiftingPositionAuto < WoodInitialLiftingPosition THEN
			IO.MotorLiftingDirection := 0;
			IF NOT Automatic.SafetyLON THEN
				Automatic.MotorL.CurrentlyMoving := TRUE;
				IO.MotorLifting := 1;
			END_IF
		ELSE
			State := 1;
			IO.MotorLifting := 0;
			Automatic.MotorL.CurrentlyMoving := FALSE;
		END_IF
	ELSIF State = 1 THEN
		IF Automatic.ExtensionPositionAuto < InitialExtensionPosition THEN
			IO.MotorExtensionDirection := 0;
			IF NOT Automatic.SafetyEON THEN
				Automatic.MotorE.CurrentlyMoving := TRUE;
				IO.MotorExtension := 1;
			END_IF
		ELSE
			State := 2;
			IO.MotorExtension := 0;
			Automatic.MotorE.CurrentlyMoving := FALSE;
		END_IF
	ELSIF State = 2 THEN
		IF Automatic.GripPositionAuto < MaxGripPosition THEN
			IO.MotorGripDirection := 0;
			IF NOT Automatic.SafetyGON THEN
				Automatic.MotorG.CurrentlyMoving := TRUE;
				IO.MotorGrip := 1;
			END_IF
		ELSE
			State := 3;
			IO.MotorGrip := 0;
			Automatic.MotorG.CurrentlyMoving := FALSE;
		END_IF
	ELSIF State = 3 THEN
		IF NOT IO.EndLiftingSensor THEN
			IO.MotorLiftingDirection := 0;
			IF NOT Automatic.SafetyLON THEN
				Automatic.MotorG.CurrentlyMoving := TRUE;
				IO.MotorLifting := 1;
			END_IF
		ELSE
			State := 4;
			IO.MotorLifting := 0;
			Automatic.MotorG.CurrentlyMoving := FALSE;
		END_IF
	ELSIF State = 4 THEN
		IF Automatic.RotationPositionAuto < RotationDropOffPosition THEN
			IO.MotorRotationDirection := 0;
			IF NOT Automatic.SafetyRON THEN
				Automatic.MotorR.CurrentlyMoving := TRUE;
				IO.MotorRotation := 1;
			END_IF
		ELSE
			State := 5;
			IO.MotorRotation := 0;
			Automatic.MotorR.CurrentlyMoving := FALSE;
		END_IF
	ELSIF State = 5 THEN
		IF NOT IO.EndExtensionSensor THEN	// it drops wood in the nearest bin
			IO.MotorExtensionDirection := 1;
			IF NOT Automatic.SafetyEON THEN
				Automatic.MotorE.CurrentlyMoving := TRUE;
				IO.MotorExtension := 1;
			END_IF
		ELSE
			State := 6;
			IO.MotorExtension := 0;
			Automatic.MotorE.CurrentlyMoving := FALSE;
		END_IF
	ELSIF State = 6 THEN
		IF NOT IO.EndGripSensor THEN
			IO.MotorGripDirection := 1;
			IF NOT Automatic.SafetyGON THEN
				Automatic.MotorG.CurrentlyMoving := TRUE;
				IO.MotorGrip := 1;
			END_IF
		ELSE
			State := 7;
			IO.MotorGrip := 0;
			Automatic.MotorG.CurrentlyMoving := FALSE;
		END_IF
	ELSIF State = 7 THEN
		IF NOT IO.EndRotationSensor THEN
			IO.MotorRotationDirection := 1;
			IF NOT Automatic.SafetyRON THEN
				Automatic.MotorR.CurrentlyMoving := TRUE;
				IO.MotorRotation := 1;
			END_IF
		ELSE
			State := 8;
			IO.MotorRotation := 0;
			Automatic.MotorR.CurrentlyMoving := FALSE;
		END_IF
	END_IF
	
	// PLASTICS:
	IF State = 8 THEN
		IF Automatic.LiftingPositionAuto < PlasticsInitialLiftingPosition THEN
			IO.MotorLiftingDirection := 0;
			IF NOT Automatic.SafetyLON THEN
				Automatic.MotorL.CurrentlyMoving := TRUE;
				IO.MotorLifting := 1;
			END_IF
		ELSE
			State := 9;
			IO.MotorLifting := 0;
			Automatic.MotorL.CurrentlyMoving := FALSE;
		END_IF
	ELSIF State = 9 THEN
		IF Automatic.ExtensionPositionAuto < InitialExtensionPosition THEN
			IO.MotorExtensionDirection := 0;
			IF NOT Automatic.SafetyEON THEN
				Automatic.MotorE.CurrentlyMoving := TRUE;
				IO.MotorExtension := 1;
			END_IF
		ELSE
			State := 10;
			IO.MotorExtension := 0;
			Automatic.MotorE.CurrentlyMoving := FALSE;
		END_IF
	ELSIF State = 10 THEN
		IF Automatic.GripPositionAuto < MaxGripPosition THEN
			IO.MotorGripDirection := 0;
			IF NOT Automatic.SafetyGON THEN
				Automatic.MotorG.CurrentlyMoving := TRUE;
				IO.MotorGrip := 1;
			END_IF
		ELSE
			State := 11;
			IO.MotorGrip := 0;
			Automatic.MotorG.CurrentlyMoving := FALSE;
		END_IF
	ELSIF State = 11 THEN
		IF NOT IO.EndLiftingSensor THEN
			IO.MotorLiftingDirection := 1;
			IF NOT Automatic.SafetyLON THEN
				Automatic.MotorL.CurrentlyMoving := TRUE;
				IO.MotorLifting := 1;
			END_IF
		ELSE
			State := 12;
			IO.MotorLifting := 0;
			Automatic.MotorL.CurrentlyMoving := FALSE;
		END_IF
	ELSIF State = 12 THEN
		IF Automatic.RotationPositionAuto < RotationDropOffPosition THEN
			IO.MotorRotationDirection := 0;
			IF NOT Automatic.SafetyRON THEN
				Automatic.MotorR.CurrentlyMoving := TRUE;
				IO.MotorRotation := 1;
			END_IF
		ELSE
			State := 13;
			IO.MotorRotation := 0;
			Automatic.MotorR.CurrentlyMoving := FALSE;
		END_IF
	ELSIF State = 13 THEN
		IF Automatic.ExtensionPositionAuto > PlasticsDropOffExtensionPosition THEN	// it drops plastics into second nearest bin
			IO.MotorExtensionDirection := 1;
			IF NOT Automatic.SafetyEON THEN
				Automatic.MotorE.CurrentlyMoving := TRUE;
				IO.MotorExtension := 1;
			END_IF
		ELSE
			State := 14;
			IO.MotorExtension := 0;
			Automatic.MotorE.CurrentlyMoving := FALSE;
		END_IF
	ELSIF State = 14 THEN
		IF NOT IO.EndGripSensor THEN
			IO.MotorGripDirection := 1;
			IF NOT Automatic.SafetyGON THEN
				Automatic.MotorG.CurrentlyMoving := TRUE;
				IO.MotorGrip := 1;
			END_IF
		ELSE
			State := 15;
			IO.MotorGrip := 0;
			Automatic.MotorG.CurrentlyMoving := FALSE;
		END_IF
	ELSIF State = 15 THEN
		IF NOT IO.EndRotationSensor THEN
			IO.MotorRotationDirection := 1;
			IF NOT Automatic.SafetyRON THEN
				Automatic.MotorR.CurrentlyMoving := TRUE;
				IO.MotorRotation := 1;
			END_IF
		ELSE
			State := 16;
			IO.MotorRotation := 0;
			Automatic.MotorR.CurrentlyMoving := FALSE;
		END_IF
	END_IF
	
	// METAL:
	IF State = 16 THEN
		IF Automatic.LiftingPositionAuto < MetalInitialLiftingPosition THEN
			IO.MotorLiftingDirection := 0;
			IF NOT Automatic.SafetyLON THEN
				Automatic.MotorL.CurrentlyMoving := TRUE;
				IO.MotorLifting := 1;
			END_IF
		ELSE
			State := 17;
			IO.MotorLifting := 0;
			Automatic.MotorL.CurrentlyMoving := FALSE;
		END_IF
	ELSIF State = 17 THEN
		IF Automatic.ExtensionPositionAuto < InitialExtensionPosition THEN
			IO.MotorExtensionDirection := 0;
			IF NOT Automatic.SafetyEON THEN
				Automatic.MotorE.CurrentlyMoving := TRUE;
				IO.MotorExtension := 1;
			END_IF
		ELSE
			State := 18;
			IO.MotorExtension := 0;
			Automatic.MotorE.CurrentlyMoving := FALSE;
		END_IF
	ELSIF State = 18 THEN
		IF Automatic.GripPositionAuto < MaxGripPosition THEN
			IO.MotorGripDirection := 0;
			IF NOT Automatic.SafetyGON THEN
				Automatic.MotorG.CurrentlyMoving := TRUE;
				IO.MotorGrip := 1;
			END_IF
		ELSE
			State := 19;
			IO.MotorGrip := 0;
			Automatic.MotorG.CurrentlyMoving := FALSE;
		END_IF
	ELSIF State = 19 THEN
		IF NOT IO.EndLiftingSensor THEN
			IO.MotorLiftingDirection := 1;
			IF NOT Automatic.SafetyLON THEN
				Automatic.MotorL.CurrentlyMoving := TRUE;
				IO.MotorLifting := 1;
			END_IF
		ELSE
			State := 20;
			IO.MotorLifting := 0;
			Automatic.MotorL.CurrentlyMoving := FALSE;
		END_IF
	ELSIF State = 20 THEN
		IF Automatic.RotationPositionAuto < RotationDropOffPosition THEN
			IO.MotorRotationDirection := 0;
			IF NOT Automatic.SafetyRON THEN
				Automatic.MotorR.CurrentlyMoving := TRUE;
				IO.MotorRotation := 1;
			END_IF
		ELSE
			State := 21;
			IO.MotorRotation := 0;
			Automatic.MotorR.CurrentlyMoving := FALSE;
		END_IF
	ELSIF State = 21 THEN
		IF Automatic.ExtensionPositionAuto > MetalDropOffExtensionPosition THEN	// it drops metal into farthest bin
			IO.MotorExtensionDirection := 1;
			IF NOT Automatic.SafetyEON THEN
				Automatic.MotorE.CurrentlyMoving := TRUE;
				IO.MotorExtension := 1;
			END_IF
		ELSE
			State := 22;
			IO.MotorExtension := 0;
			Automatic.MotorE.CurrentlyMoving := FALSE;
		END_IF
	ELSIF State = 22 THEN
		IF NOT IO.EndGripSensor THEN
			IO.MotorGripDirection := 1;
			IF NOT Automatic.SafetyGON THEN
				Automatic.MotorG.CurrentlyMoving := TRUE;
				IO.MotorGrip := 1;
			END_IF
		ELSE
			State := 23;
			IO.MotorGrip := 0;
			Automatic.MotorG.CurrentlyMoving := FALSE;
		END_IF
	ELSIF State = 23 THEN
		IF NOT IO.EndRotationSensor THEN
			IO.MotorRotationDirection := 1;
			IF NOT Automatic.SafetyRON THEN
				Automatic.MotorR.CurrentlyMoving := TRUE;
				IO.MotorRotation := 1;
			END_IF
		ELSE
			State := 24;
			IO.MotorRotation := 0;
			Automatic.MotorR.CurrentlyMoving := FALSE;
		END_IF
	ELSIF State = 24 THEN
		SuccesfullyEnded := TRUE;
		State := 0;
		RETURN;
	END_IF
END_IF
RETURN;

END_FUNCTION_BLOCK

// ---- POUs/Motor.TcPOU
FUNCTION_BLOCK PUBLIC Motor
VAR_INPUT
	CurrentlyMoving: BOOL;	// we need this because stepSwitches can be 1 and we should not move
	// Current position is currently stored in the Automatic GVLs.
END_VAR
VAR_OUTPUT
END_VAR
VAR
	
END_VAR

END_FUNCTION_BLOCK

// ---- POUs/CountCurrentPosition.TcPOU
PROGRAM CountCurrentPosition
VAR
END_VAR

// ONLY COUNTING, NO SETTING MOTORS ON/OFF

// COUNT ROTATION:
IF IO.Initialized AND IO.StepRotatonSwitch = 1 THEN
	IO.LEDGreen := 0;
	IF IO.MotorRotationDirection = 0 THEN
		IF Automatic.MotorR.CurrentlyMoving THEN
			Automatic.RotationPositionCurrent := Automatic.RotationPositionCurrent + 1;
		ELSIF NOT IO.Switch THEN
			Automatic.RotationPositionAuto := Automatic.RotationPositionAuto + 1;
			Automatic.RotationPositionCurrent := Automatic.RotationPositionCurrent + 1;
		END_IF
	ELSE
		IF Automatic.MotorR.CurrentlyMoving THEN
			Automatic.RotationPositionCurrent := Automatic.RotationPositionCurrent - 1;
		ELSIF NOT IO.Switch THEN
			Automatic.RotationPositionAuto := Automatic.RotationPositionAuto - 1;
			Automatic.RotationPositionCurrent := Automatic.RotationPositionCurrent - 1;
		END_IF
	END_IF
ELSE
	IO.LEDGreen := 1;
END_IF

// COUNT Extension:
IF IO.Initialized AND IO.StepExtensionSwitch = 1 THEN
	IO.LEDGreen := 0;
	IF IO.MotorExtensionDirection = 0 THEN
		IF Automatic.MotorE.CurrentlyMoving THEN
			Automatic.ExtensionPositionCurrent := Automatic.ExtensionPositionCurrent + 1;
		ELSIF NOT IO.Switch THEN
			Automatic.ExtensionPositionAuto := Automatic.ExtensionPositionAuto + 1;
			Automatic.ExtensionPositionCurrent := Automatic.ExtensionPositionCurrent + 1;
		END_IF
	ELSE
		IF Automatic.MotorE.CurrentlyMoving THEN
			Automatic.ExtensionPositionCurrent := Automatic.ExtensionPositionCurrent - 1;
		ELSIF NOT IO.Switch THEN
			Automatic.ExtensionPositionAuto := Automatic.ExtensionPositionAuto - 1;
			Automatic.ExtensionPositionCurrent := Automatic.ExtensionPositionCurrent - 1;
		END_IF
	END_IF
ELSE
	IO.LEDGreen := 1;
END_IF

// COUNT Lifting:
IF IO.Initialized AND IO.StepLiftingSwitch = 1 THEN
	IO.LEDGreen := 0;
	IF IO.MotorLiftingDirection = 0 THEN
		IF Automatic.MotorL.CurrentlyMoving THEN
			Automatic.LiftingPositionCurrent := Automatic.LiftingPositionCurrent + 1;
		ELSIF NOT IO.Switch THEN
			Automatic.LiftingPositionAuto := Automatic.LiftingPositionAuto + 1;
			Automatic.LiftingPositionCurrent := Automatic.LiftingPositionCurrent + 1;
		END_IF
	ELSE
		IF Automatic.MotorL.CurrentlyMoving THEN
			Automatic.LiftingPositionCurrent := Automatic.LiftingPositionCurrent - 1;
		ELSIF NOT IO.Switch THEN
			Automatic.LiftingPositionAuto := Automatic.LiftingPositionAuto - 1;
			Automatic.LiftingPositionCurrent := Automatic.LiftingPositionCurrent - 1;
		END_IF
	END_IF
ELSE
	IO.LEDGreen := 1;
END_IF

// COUNT Grip:
IF IO.Initialized AND IO.StepGripSwitch = 1 THEN
	IO.LEDGreen := 0;
	IF IO.MotorGripDirection = 0 THEN
		IF NOT IO.Switch AND Automatic.MotorG.CurrentlyMoving THEN
			Automatic.GripPositionAuto := Automatic.GripPositionAuto + 1;
			Automatic.GripPositionCurrent := Automatic.GripPositionCurrent + 1;
		ELSIF Automatic.MotorG.CurrentlyMoving THEN
			Automatic.GripPositionCurrent := Automatic.GripPositionCurrent + 1;
		END_IF
	ELSE
		IF NOT IO.Switch AND Automatic.MotorG.CurrentlyMoving THEN
			Automatic.GripPositionAuto := Automatic.GripPositionAuto - 1;
			Automatic.GripPositionCurrent := Automatic.GripPositionCurrent - 1;
		ELSIF Automatic.MotorG.CurrentlyMoving THEN
			Automatic.GripPositionCurrent := Automatic.GripPositionCurrent - 1;
		END_IF
	END_IF
ELSE
	IO.LEDGreen := 1;
END_IF

END_PROGRAM

// ---- POUs/Recipe11.TcPOU
PROGRAM Recipe13
VAR_INPUT
	ExecutingRecipe1: BOOL;
END_VAR
VAR_OUTPUT
	SuccesfullyEnded: BOOL := FALSE;
END_VAR
VAR
	State: INT := 0;
	WoodInitialLiftingPosition: INT := 50;
	InitialExtensionPosition: INT := 388;
	MaxGripPosition: INT := 160;
	RotationDropOffPosition: INT := 300;
	PlasticsInitialLiftingPosition: INT := 250;
	PlasticsDropOffExtensionPosition: INT := 300;
	MetalInitialLiftingPosition: INT := 400;
	MetalDropOffExtensionPosition: INT := 500;
END_VAR

// Recipe is sequence of moves to execute the task.

IF ExecutingRecipe1 THEN	// we start executing recipe1 (again)
	SuccesfullyEnded := FALSE;
END_IF

IF NOT IO.Switch AND NOT SuccesfullyEnded THEN
	IO.LEDGreen := 1;
	// WOOD:
	IF State = 0 THEN
		IF Automatic.LiftingPositionAuto < WoodInitialLiftingPosition THEN
			IO.MotorLiftingDirection := 0;
			IF NOT Automatic.SafetyLON THEN
				Automatic.MotorL.CurrentlyMoving := TRUE;
				IO.MotorLifting := 1;
			END_IF
		ELSE
			State := 1;
			IO.MotorLifting := 0;
			Automatic.MotorL.CurrentlyMoving := FALSE;
		END_IF
	ELSIF State = 1 THEN
		IF Automatic.ExtensionPositionAuto < InitialExtensionPosition THEN
			IO.MotorExtensionDirection := 0;
			IF NOT Automatic.SafetyEON THEN
				Automatic.MotorE.CurrentlyMoving := TRUE;
				IO.MotorExtension := 1;
			END_IF
		ELSE
			State := 2;
			IO.MotorExtension := 0;
			Automatic.MotorE.CurrentlyMoving := FALSE;
		END_IF
	ELSIF State = 2 THEN
		IF Automatic.GripPositionAuto < MaxGripPosition THEN
			IO.MotorGripDirection := 0;
			IF NOT Automatic.SafetyGON THEN
				Automatic.MotorG.CurrentlyMoving := TRUE;
				IO.MotorGrip := 1;
			END_IF
		ELSE
			State := 3;
			IO.MotorGrip := 0;
			Automatic.MotorG.CurrentlyMoving := FALSE;
		END_IF
	ELSIF State = 3 THEN
		IF NOT IO.EndLiftingSensor THEN
			IO.MotorLiftingDirection := 1;
			IF NOT Automatic.SafetyLON THEN
				Automatic.MotorG.CurrentlyMoving := TRUE;
				IO.MotorLifting := 1;
			END_IF
		ELSE
			State := 4;
			IO.MotorLifting := 0;
			Automatic.MotorL.CurrentlyMoving := FALSE;
		END_IF
	ELSIF State = 4 THEN
		IF Automatic.RotationPositionAuto < RotationDropOffPosition THEN
			IO.MotorRotationDirection := 0;
			IF NOT Automatic.SafetyRON THEN
				Automatic.MotorR.CurrentlyMoving := TRUE;
				IO.MotorRotation := 1;
			END_IF
		ELSE
			State := 5;
			IO.MotorRotation := 0;
			Automatic.MotorR.CurrentlyMoving := FALSE;
		END_IF
	ELSIF State = 5 THEN
		IF NOT IO.EndExtensionSensor THEN	// it drops wood in the nearest bin
			IO.MotorExtensionDirection := 1;
			IF NOT Automatic.SafetyEON THEN
				Automatic.MotorE.CurrentlyMoving := TRUE;
				IO.MotorExtension := 1;
			END_IF
		ELSE
			State := 6;
			IO.MotorExtension := 0;
			Automatic.MotorE.CurrentlyMoving := FALSE;
		END_IF
	ELSIF State = 6 THEN
		IF NOT IO.EndGripSensor THEN
			IO.MotorGripDirection := 1;
			IF NOT Automatic.SafetyGON THEN
				Automatic.MotorG.CurrentlyMoving := TRUE;
				IO.MotorGrip := 1;
			END_IF
		ELSE
			State := 7;
			IO.MotorGrip := 0;
			Automatic.MotorG.CurrentlyMoving := FALSE;
		END_IF
	ELSIF State = 7 THEN
		IF NOT IO.EndRotationSensor THEN
			IO.MotorRotationDirection := 1;
			IF NOT Automatic.SafetyRON THEN
				Automatic.MotorR.CurrentlyMoving := TRUE;
				IO.MotorRotation := 1;
			END_IF
		ELSE
			State := 8;
			IO.MotorRotation := 0;
			Automatic.MotorR.CurrentlyMoving := FALSE;
		END_IF
	END_IF
	
	// PLASTICS:
	IF State = 8 THEN
		IF Automatic.LiftingPositionAuto < PlasticsInitialLiftingPosition THEN
			IO.MotorLiftingDirection := 0;
			IF NOT Automatic.SafetyLON THEN
				Automatic.MotorL.CurrentlyMoving := TRUE;
				IO.MotorLifting := 1;
			END_IF
		ELSE
			State := 9;
			IO.MotorLifting := 0;
			Automatic.MotorL.CurrentlyMoving := FALSE;
		END_IF
	ELSIF State = 9 THEN
		IF Automatic.ExtensionPositionAuto < InitialExtensionPosition THEN
			IO.MotorExtensionDirection := 0;
			IF NOT Automatic.SafetyEON THEN
				Automatic.MotorE.CurrentlyMoving := TRUE;
				IO.MotorExtension := 1;
			END_IF
		ELSE
			State := 10;
			IO.MotorExtension := 0;
			Automatic.MotorE.CurrentlyMoving := FALSE;
		END_IF
	ELSIF State = 10 THEN
		IF Automatic.GripPositionAuto < MaxGripPosition THEN
			IO.MotorGripDirection := 0;
			IF NOT Automatic.SafetyGON THEN
				Automatic.MotorG.CurrentlyMoving := TRUE;
				IO.MotorGrip := 1;
			END_IF
		ELSE
			State := 11;
			IO.MotorGrip := 0;
			Automatic.MotorG.CurrentlyMoving := FALSE;
		END_IF
	ELSIF State = 11 THEN
		IF NOT IO.EndLiftingSensor THEN
			IO.MotorLiftingDirection := 1;
			IF NOT Automatic.SafetyLON THEN
				Automatic.MotorL.CurrentlyMoving := TRUE;
				IO.MotorLifting := 1;
			END_IF
		ELSE
			State := 12;
			IO.MotorLifting := 0;
			Automatic.MotorL.CurrentlyMoving := FALSE;
		END_IF
	ELSIF State = 12 THEN
		IF Automatic.RotationPositionAuto < RotationDropOffPosition THEN
			IO.MotorRotationDirection := 0;
			IF NOT Automatic.SafetyRON THEN
				Automatic.MotorR.CurrentlyMoving := TRUE;
				IO.MotorRotation := 1;
			END_IF
		ELSE
			State := 13;
			IO.MotorRotation := 0;
			Automatic.MotorR.CurrentlyMoving := FALSE;
		END_IF
	ELSIF State = 13 THEN
		IF Automatic.ExtensionPositionAuto > PlasticsDropOffExtensionPosition THEN	// it drops plastics into second nearest bin
			IO.MotorExtensionDirection := 1;
			IF NOT Automatic.SafetyEON THEN
				Automatic.MotorE.CurrentlyMoving := TRUE;
				IO.MotorExtension := 1;
			END_IF
		ELSE
			State := 14;
			IO.MotorExtension := 0;
			Automatic.MotorE.CurrentlyMoving := FALSE;
		END_IF
	ELSIF State = 14 THEN
		IF NOT IO.EndGripSensor THEN
			IO.MotorGripDirection := 1;
			IF NOT Automatic.SafetyGON THEN
				Automatic.MotorG.CurrentlyMoving := TRUE;
				IO.MotorGrip := 1;
			END_IF
		ELSE
			State := 15;
			IO.MotorGrip := 0;
			Automatic.MotorG.CurrentlyMoving := FALSE;
		END_IF
	ELSIF State = 15 THEN
		IF NOT IO.EndRotationSensor THEN
			IO.MotorRotationDirection := 1;
			IF NOT Automatic.SafetyRON THEN
				Automatic.MotorR.CurrentlyMoving := TRUE;
				IO.MotorRotation := 1;
			END_IF
		ELSE
			State := 16;
			IO.MotorRotation := 0;
			Automatic.MotorR.CurrentlyMoving := FALSE;
		END_IF
	END_IF
	
	// METAL:
	IF State = 16 THEN
		IF Automatic.LiftingPositionAuto < MetalInitialLiftingPosition THEN
			IO.MotorLiftingDirection := 0;
			IF NOT Automatic.SafetyLON THEN
				Automatic.MotorL.CurrentlyMoving := TRUE;
				IO.MotorLifting := 1;
			END_IF
		ELSE
			State := 17;
			IO.MotorLifting := 0;
			Automatic.MotorL.CurrentlyMoving := FALSE;
		END_IF
	ELSIF State = 17 THEN
		IF Automatic.ExtensionPositionAuto < InitialExtensionPosition THEN
			IO.MotorExtensionDirection := 0;
			IF NOT Automatic.SafetyEON THEN
				Automatic.MotorE.CurrentlyMoving := TRUE;
				IO.MotorExtension := 1;
			END_IF
		ELSE
			State := 18;
			IO.MotorExtension := 0;
			Automatic.MotorE.CurrentlyMoving := FALSE;
		END_IF
	ELSIF State = 18 THEN
		IF Automatic.GripPositionAuto < MaxGripPosition THEN
			IO.MotorGripDirection := 0;
			IF NOT Automatic.SafetyGON THEN
				Automatic.MotorG.CurrentlyMoving := TRUE;
				IO.MotorGrip := 1;
			END_IF
		ELSE
			State := 19;
			IO.MotorGrip := 0;
			Automatic.MotorG.CurrentlyMoving := FALSE;
		END_IF
	ELSIF State = 19 THEN
		IF NOT IO.EndLiftingSensor THEN
			IO.MotorLiftingDirection := 1;
			IF NOT Automatic.SafetyLON THEN
				Automatic.MotorL.CurrentlyMoving := TRUE;
				IO.MotorLifting := 1;
			END_IF
		ELSE
			State := 20;
			IO.MotorLifting := 0;
			Automatic.MotorL.CurrentlyMoving := FALSE;
		END_IF
	ELSIF State = 20 THEN
		IF Automatic.RotationPositionAuto < RotationDropOffPosition THEN
			IO.MotorRotationDirection := 0;
			IF NOT Automatic.SafetyRON THEN
				Automatic.MotorR.CurrentlyMoving := TRUE;
				IO.MotorRotation := 1;
			END_IF
		ELSE
			State := 21;
			IO.MotorRotation := 0;
			Automatic.MotorR.CurrentlyMoving := FALSE;
		END_IF
	ELSIF State = 21 THEN
		IF Automatic.ExtensionPositionAuto > MetalDropOffExtensionPosition THEN	// it drops metal into farthest bin
			IO.MotorExtensionDirection := 1;
			IF NOT Automatic.SafetyEON THEN
				Automatic.MotorE.CurrentlyMoving := TRUE;
				IO.MotorExtension := 1;
			END_IF
		ELSE
			State := 22;
			IO.MotorExtension := 0;
			Automatic.MotorE.CurrentlyMoving := FALSE;
		END_IF
	ELSIF State = 22 THEN
		IF NOT IO.EndGripSensor THEN
			IO.MotorGripDirection := 1;
			IF NOT Automatic.SafetyGON THEN
				Automatic.MotorG.CurrentlyMoving := TRUE;
				IO.MotorGrip := 1;
			END_IF
		ELSE
			State := 23;
			IO.MotorGrip := 0;
			Automatic.MotorG.CurrentlyMoving := FALSE;
		END_IF
	ELSIF State = 23 THEN
		IF NOT IO.EndRotationSensor THEN
			IO.MotorRotationDirection := 1;
			IF NOT Automatic.SafetyRON THEN
				Automatic.MotorR.CurrentlyMoving := TRUE;
				IO.MotorRotation := 1;
			END_IF
		ELSE
			State := 24;
			IO.MotorRotation := 0;
			Automatic.MotorR.CurrentlyMoving := FALSE;
		END_IF
	ELSIF State = 24 THEN
		SuccesfullyEnded := TRUE;
		State := 0;
		RETURN;
	END_IF
END_IF
RETURN;

END_PROGRAM

// ---- POUs/Recipe13.TcPOU
PROGRAM Recipe13
VAR_INPUT
	ExecutingRecipe1: BOOL;
END_VAR
VAR_OUTPUT
	SuccesfullyEnded: BOOL := FALSE;
END_VAR
VAR
	State: INT := 0;
	WoodInitialLiftingPosition: INT := 50;
	InitialExtensionPosition: INT := 388;
	MaxGripPosition: INT := 160;
	RotationDropOffPosition: INT := 300;
	PlasticsInitialLiftingPosition: INT := 250;
	PlasticsDropOffExtensionPosition: INT := 300;
	MetalInitialLiftingPosition: INT := 400;
	MetalDropOffExtensionPosition: INT := 500;
END_VAR

// Recipe is sequence of moves to execute the task.

IF ExecutingRecipe1 THEN	// we start executing recipe1 (again)
	SuccesfullyEnded := FALSE;
END_IF

IF NOT IO.Switch AND NOT SuccesfullyEnded THEN
	IO.LEDGreen := 1;
	// WOOD:
	IF State = 0 THEN
		IF Automatic.LiftingPositionAuto < WoodInitialLiftingPosition THEN
			IO.MotorLiftingDirection := 0;
			IF NOT Automatic.SafetyLON THEN
				Automatic.MotorL.CurrentlyMoving := TRUE;
				IO.MotorLifting := 1;
			END_IF
		ELSE
			State := 1;
			IO.MotorLifting := 0;
			Automatic.MotorL.CurrentlyMoving := FALSE;
		END_IF
	ELSIF State = 1 THEN
		IF Automatic.ExtensionPositionAuto < InitialExtensionPosition THEN
			IO.MotorExtensionDirection := 0;
			IF NOT Automatic.SafetyEON THEN
				Automatic.MotorE.CurrentlyMoving := TRUE;
				IO.MotorExtension := 1;
			END_IF
		ELSE
			State := 2;
			IO.MotorExtension := 0;
			Automatic.MotorE.CurrentlyMoving := FALSE;
		END_IF
	ELSIF State = 2 THEN
		IF Automatic.GripPositionAuto < MaxGripPosition THEN
			IO.MotorGripDirection := 0;
			IF NOT Automatic.SafetyGON THEN
				Automatic.MotorG.CurrentlyMoving := TRUE;
				IO.MotorGrip := 1;
			END_IF
		ELSE
			State := 3;
			IO.MotorGrip := 0;
			Automatic.MotorG.CurrentlyMoving := FALSE;
		END_IF
	ELSIF State = 3 THEN
		IF NOT IO.EndLiftingSensor THEN
			IO.MotorLiftingDirection := 1;
			IF NOT Automatic.SafetyLON THEN
				Automatic.MotorG.CurrentlyMoving := TRUE;
				IO.MotorLifting := 1;
			END_IF
		ELSE
			State := 4;
			IO.MotorLifting := 0;
			Automatic.MotorL.CurrentlyMoving := FALSE;
		END_IF
	ELSIF State = 4 THEN
		IF Automatic.RotationPositionAuto < RotationDropOffPosition THEN
			IO.MotorRotationDirection := 0;
			IF NOT Automatic.SafetyRON THEN
				Automatic.MotorR.CurrentlyMoving := TRUE;
				IO.MotorRotation := 1;
			END_IF
		ELSE
			State := 5;
			IO.MotorRotation := 0;
			Automatic.MotorR.CurrentlyMoving := FALSE;
		END_IF
	ELSIF State = 5 THEN
		IF NOT IO.EndExtensionSensor THEN	// it drops wood in the nearest bin
			IO.MotorExtensionDirection := 1;
			IF NOT Automatic.SafetyEON THEN
				Automatic.MotorE.CurrentlyMoving := TRUE;
				IO.MotorExtension := 1;
			END_IF
		ELSE
			State := 6;
			IO.MotorExtension := 0;
			Automatic.MotorE.CurrentlyMoving := FALSE;
		END_IF
	ELSIF State = 6 THEN
		IF NOT IO.EndGripSensor THEN
			IO.MotorGripDirection := 1;
			IF NOT Automatic.SafetyGON THEN
				Automatic.MotorG.CurrentlyMoving := TRUE;
				IO.MotorGrip := 1;
			END_IF
		ELSE
			State := 7;
			IO.MotorGrip := 0;
			Automatic.MotorG.CurrentlyMoving := FALSE;
		END_IF
	ELSIF State = 7 THEN
		IF NOT IO.EndRotationSensor THEN
			IO.MotorRotationDirection := 1;
			IF NOT Automatic.SafetyRON THEN
				Automatic.MotorR.CurrentlyMoving := TRUE;
				IO.MotorRotation := 1;
			END_IF
		ELSE
			State := 8;
			IO.MotorRotation := 0;
			Automatic.MotorR.CurrentlyMoving := FALSE;
		END_IF
	END_IF
	
	// PLASTICS:
	IF State = 8 THEN
		IF Automatic.LiftingPositionAuto < PlasticsInitialLiftingPosition THEN
			IO.MotorLiftingDirection := 0;
			IF NOT Automatic.SafetyLON THEN
				Automatic.MotorL.CurrentlyMoving := TRUE;
				IO.MotorLifting := 1;
			END_IF
		ELSE
			State := 9;
			IO.MotorLifting := 0;
			Automatic.MotorL.CurrentlyMoving := FALSE;
		END_IF
	ELSIF State = 9 THEN
		IF Automatic.ExtensionPositionAuto < InitialExtensionPosition THEN
			IO.MotorExtensionDirection := 0;
			IF NOT Automatic.SafetyEON THEN
				Automatic.MotorE.CurrentlyMoving := TRUE;
				IO.MotorExtension := 1;
			END_IF
		ELSE
			State := 10;
			IO.MotorExtension := 0;
			Automatic.MotorE.CurrentlyMoving := FALSE;
		END_IF
	ELSIF State = 10 THEN
		IF Automatic.GripPositionAuto < MaxGripPosition THEN
			IO.MotorGripDirection := 0;
			IF NOT Automatic.SafetyGON THEN
				Automatic.MotorG.CurrentlyMoving := TRUE;
				IO.MotorGrip := 1;
			END_IF
		ELSE
			State := 11;
			IO.MotorGrip := 0;
			Automatic.MotorG.CurrentlyMoving := FALSE;
		END_IF
	ELSIF State = 11 THEN
		IF NOT IO.EndLiftingSensor THEN
			IO.MotorLiftingDirection := 1;
			IF NOT Automatic.SafetyLON THEN
				Automatic.MotorL.CurrentlyMoving := TRUE;
				IO.MotorLifting := 1;
			END_IF
		ELSE
			State := 12;
			IO.MotorLifting := 0;
			Automatic.MotorL.CurrentlyMoving := FALSE;
		END_IF
	ELSIF State = 12 THEN
		IF Automatic.RotationPositionAuto < RotationDropOffPosition THEN
			IO.MotorRotationDirection := 0;
			IF NOT Automatic.SafetyRON THEN
				Automatic.MotorR.CurrentlyMoving := TRUE;
				IO.MotorRotation := 1;
			END_IF
		ELSE
			State := 13;
			IO.MotorRotation := 0;
			Automatic.MotorR.CurrentlyMoving := FALSE;
		END_IF
	ELSIF State = 13 THEN
		IF Automatic.ExtensionPositionAuto > PlasticsDropOffExtensionPosition THEN	// it drops plastics into second nearest bin
			IO.MotorExtensionDirection := 1;
			IF NOT Automatic.SafetyEON THEN
				Automatic.MotorE.CurrentlyMoving := TRUE;
				IO.MotorExtension := 1;
			END_IF
		ELSE
			State := 14;
			IO.MotorExtension := 0;
			Automatic.MotorE.CurrentlyMoving := FALSE;
		END_IF
	ELSIF State = 14 THEN
		IF NOT IO.EndGripSensor THEN
			IO.MotorGripDirection := 1;
			IF NOT Automatic.SafetyGON THEN
				Automatic.MotorG.CurrentlyMoving := TRUE;
				IO.MotorGrip := 1;
			END_IF
		ELSE
			State := 15;
			IO.MotorGrip := 0;
			Automatic.MotorG.CurrentlyMoving := FALSE;
		END_IF
	ELSIF State = 15 THEN
		IF NOT IO.EndRotationSensor THEN
			IO.MotorRotationDirection := 1;
			IF NOT Automatic.SafetyRON THEN
				Automatic.MotorR.CurrentlyMoving := TRUE;
				IO.MotorRotation := 1;
			END_IF
		ELSE
			State := 16;
			IO.MotorRotation := 0;
			Automatic.MotorR.CurrentlyMoving := FALSE;
		END_IF
	END_IF
	
	// METAL:
	IF State = 16 THEN
		IF Automatic.LiftingPositionAuto < MetalInitialLiftingPosition THEN
			IO.MotorLiftingDirection := 0;
			IF NOT Automatic.SafetyLON THEN
				Automatic.MotorL.CurrentlyMoving := TRUE;
				IO.MotorLifting := 1;
			END_IF
		ELSE
			State := 17;
			IO.MotorLifting := 0;
			Automatic.MotorL.CurrentlyMoving := FALSE;
		END_IF
	ELSIF State = 17 THEN
		IF Automatic.ExtensionPositionAuto < InitialExtensionPosition THEN
			IO.MotorExtensionDirection := 0;
			IF NOT Automatic.SafetyEON THEN
				Automatic.MotorE.CurrentlyMoving := TRUE;
				IO.MotorExtension := 1;
			END_IF
		ELSE
			State := 18;
			IO.MotorExtension := 0;
			Automatic.MotorE.CurrentlyMoving := FALSE;
		END_IF
	ELSIF State = 18 THEN
		IF Automatic.GripPositionAuto < MaxGripPosition THEN
			IO.MotorGripDirection := 0;
			IF NOT Automatic.SafetyGON THEN
				Automatic.MotorG.CurrentlyMoving := TRUE;
				IO.MotorGrip := 1;
			END_IF
		ELSE
			State := 19;
			IO.MotorGrip := 0;
			Automatic.MotorG.CurrentlyMoving := FALSE;
		END_IF
	ELSIF State = 19 THEN
		IF NOT IO.EndLiftingSensor THEN
			IO.MotorLiftingDirection := 1;
			IF NOT Automatic.SafetyLON THEN
				Automatic.MotorL.CurrentlyMoving := TRUE;
				IO.MotorLifting := 1;
			END_IF
		ELSE
			State := 20;
			IO.MotorLifting := 0;
			Automatic.MotorL.CurrentlyMoving := FALSE;
		END_IF
	ELSIF State = 20 THEN
		IF Automatic.RotationPositionAuto < RotationDropOffPosition THEN
			IO.MotorRotationDirection := 0;
			IF NOT Automatic.SafetyRON THEN
				Automatic.MotorR.CurrentlyMoving := TRUE;
				IO.MotorRotation := 1;
			END_IF
		ELSE
			State := 21;
			IO.MotorRotation := 0;
			Automatic.MotorR.CurrentlyMoving := FALSE;
		END_IF
	ELSIF State = 21 THEN
		IF Automatic.ExtensionPositionAuto > MetalDropOffExtensionPosition THEN	// it drops metal into farthest bin
			IO.MotorExtensionDirection := 1;
			IF NOT Automatic.SafetyEON THEN
				Automatic.MotorE.CurrentlyMoving := TRUE;
				IO.MotorExtension := 1;
			END_IF
		ELSE
			State := 22;
			IO.MotorExtension := 0;
			Automatic.MotorE.CurrentlyMoving := FALSE;
		END_IF
	ELSIF State = 22 THEN
		IF NOT IO.EndGripSensor THEN
			IO.MotorGripDirection := 1;
			IF NOT Automatic.SafetyGON THEN
				Automatic.MotorG.CurrentlyMoving := TRUE;
				IO.MotorGrip := 1;
			END_IF
		ELSE
			State := 23;
			IO.MotorGrip := 0;
			Automatic.MotorG.CurrentlyMoving := FALSE;
		END_IF
	ELSIF State = 23 THEN
		IF NOT IO.EndRotationSensor THEN
			IO.MotorRotationDirection := 1;
			IF NOT Automatic.SafetyRON THEN
				Automatic.MotorR.CurrentlyMoving := TRUE;
				IO.MotorRotation := 1;
			END_IF
		ELSE
			State := 24;
			IO.MotorRotation := 0;
			Automatic.MotorR.CurrentlyMoving := FALSE;
		END_IF
	ELSIF State = 24 THEN
		SuccesfullyEnded := TRUE;
		State := 0;
		RETURN;
	END_IF
END_IF
RETURN;

END_PROGRAM
